TYPE TcoGenericInterpolatorHw :
STRUCT
	// In
	Inputs : TcoGenericInterpolatorHwInputs;

	// Out					
	Outputs : TcoGenericInterpolatorHwOutputs;
END_STRUCT
END_TYPE

(* stored: Version 1.1.0.1, ProductVersion 3.1.4024.12
   DUT TcoGenericInterpolatorHw: Id {49fa38fe-8868-4245-bf80-1b12392b3135} *)
